FUNCTION_BLOCK CM_DoorLock EXTENDS CM_Base //--IMPLEMENTS I_Door
VAR_INPUT
	i_stSettings : ST_SettingsDoorLock;
END_VAR
VAR
	// Inputs
	I_bStaDoorIsClosed AT %I* : BOOL; // Door is closed
	I_bStaLockIsReleased AT %I* : BOOL; // Lock is released
	
	// Outputs
	Q_bCmdReleaseLock AT %Q* : BOOL; // FALSE = Apply, TRUE = Release
			
	// Requests
	s_bReqReleaseLock : BOOL;
	s_bReqApplyLock : BOOL;
	
	//----------------------Properties---------------------------//
	// States
	s_bStaDoorIsClosed : BOOL;
	s_bStaDoorIsOpened : BOOL;
	s_bStaLockIsApplied : BOOL;
	s_bStaLockIsReleased : BOOL;
	s_bCfgAutoLockAtClosing : BOOL;
	
	// Timers
	s_tonReleasingLockTimeout : TON;
	s_tonApplyingLockTimeout : TON;
	
	// Alarms
	s_fbAlarmHandlerReleasingLockTimeout : FB_AlarmHandler;
	s_fbAlarmHandlerApplyingLockTimeout : FB_AlarmHandler;
	s_fbAlarmHandlerDoorIsNotClosed : FB_AlarmHandler;
	
	s_errLockReleasingTimeout : BOOL;
	s_errLockApplyingTimeout : BOOL;
	s_wrnDoorIsNotClosed : BOOL;
		
	s_bStaDoorIsClosedOsr : R_TRIG; 
END_VAR


SUPER^();

METHOD PROTECTED _m_Alarms : BOOL

IF NOT SUPER^._m_Alarms() THEN
	RETURN;
END_IF

// Timeout (timers)
s_tonReleasingLockTimeout(
	IN := i_bReqEnable AND s_bReqReleaseLock AND NOT(s_bStaLockIsReleased),
	PT := i_stSettings.tReleasingLockTimeout);
	
s_tonApplyingLockTimeout(
	IN := i_bReqEnable AND s_bReqApplyLock AND NOT(s_bStaLockIsApplied),
	PT := i_stSettings.tApplyingLockTimeout);

// Set error bits
s_errLockReleasingTimeout := (s_tonReleasingLockTimeout.Q OR s_errLockReleasingTimeout) AND NOT(i_bCmdReset);
s_errLockApplyingTimeout := (s_tonApplyingLockTimeout.Q OR s_errLockApplyingTimeout) AND NOT(i_bCmdReset);

// Alarm Handlers
s_fbAlarmHandlerReleasingLockTimeout(
	i_bStaActive := s_errLockReleasingTimeout,
	i_eAlarmLevel := E_AlarmLevel.Alarm,
	i_sAlarmText := CONCAT(i_sCmName , ': Lock - releasing timeout.') );
	
s_fbAlarmHandlerApplyingLockTimeout(
	i_bStaActive := s_errLockApplyingTimeout,
	i_eAlarmLevel := E_AlarmLevel.Alarm,
	i_sAlarmText := CONCAT(i_sCmName , ': Lock - applying timeout.') );
	
s_fbAlarmHandlerDoorIsNotClosed(
	i_bStaActive := s_wrnDoorIsNotClosed,
	i_eAlarmLevel := E_AlarmLevel.Warning,
	i_sAlarmText := CONCAT(i_sCmName , ': Door - not closed (close door before lock can be applied).') );	
	
// Alarm collector	
s_bStaError := 
	s_fbAlarmHandlerReleasingLockTimeout.q_bStaActive
	OR s_fbAlarmHandlerApplyingLockTimeout.q_bStaActive;

_m_Alarms := TRUE;
END_METHOD

METHOD PROTECTED _m_Devices : BOOL

IF NOT SUPER^._m_Devices() THEN
	RETURN;
END_IF

IF s_bStaError THEN
	s_bReqReleaseLock := FALSE;
	s_bReqApplyLock := FALSE;
END_IF
	
IF s_bCfgAutoLockAtClosing AND s_bStaDoorIsClosedOsr.Q THEN
	s_bReqReleaseLock := FALSE;
	s_bReqApplyLock := TRUE;
END_IF

IF s_bStaDoorIsClosed THEN
	s_wrnDoorIsNotClosed := FALSE;	
END_IF

_m_Devices := TRUE;
END_METHOD

METHOD PROTECTED _m_Hmi : BOOL

IF NOT SUPER^._m_Hmi() THEN
	RETURN;
END_IF

_m_Hmi := TRUE;
END_METHOD

METHOD PROTECTED _m_Init : BOOL

IF NOT SUPER^._m_Init() THEN
	RETURN;
END_IF

_m_Init := TRUE;
END_METHOD

METHOD PROTECTED _m_Inputs : BOOL

IF NOT SUPER^._m_Inputs() THEN
	RETURN;
END_IF

s_bStaLockIsReleased := I_bStaLockIsReleased;
s_bStaLockIsApplied := NOT(I_bStaLockIsReleased);
s_bStaDoorIsClosed := I_bStaDoorIsClosed;
s_bStaDoorIsOpened := NOT(I_bStaDoorIsClosed);

s_bStaDoorIsClosedOsr(CLK := s_bStaDoorIsClosed);

_m_Inputs := TRUE;
END_METHOD

METHOD PROTECTED _m_Outputs : BOOL

IF NOT SUPER^._m_Outputs() THEN
	RETURN;
END_IF

Q_bCmdReleaseLock := s_bReqReleaseLock;

_m_Outputs := TRUE;
END_METHOD

/// Request to apply door-lock (only if door is closed)
METHOD PUBLIC m_Apply : BOOL

IF NOT i_bReqEnable THEN 
	RETURN;
END_IF

IF s_bStaDoorIsClosed THEN
	s_bReqReleaseLock := FALSE;
	s_bReqApplyLock := TRUE;
ELSE
	s_wrnDoorIsNotClosed := TRUE;	
END_IF
	
m_Apply := TRUE;
END_METHOD

/// Request to release door-lock
METHOD PUBLIC m_Release : BOOL

IF NOT i_bReqEnable THEN 
	RETURN;
END_IF

s_bReqReleaseLock := TRUE;
s_bReqApplyLock := FALSE;
s_wrnDoorIsNotClosed := FALSE;

m_Release := TRUE;
END_METHOD

{attribute 'monitoring':='call'}
PROPERTY PUBLIC p_bCfgAutoLockAtClosing : BOOL
GET

p_bCfgAutoLockAtClosing := s_bCfgAutoLockAtClosing;
END_GET
SET

s_bCfgAutoLockAtClosing := p_bCfgAutoLockAtClosing;
END_SET
END_PROPERTY

{attribute 'monitoring':='call'}
PROPERTY PUBLIC p_bStaDoorIsClosed : BOOL
GET

p_bStaDoorIsClosed := s_bStaDoorIsClosed;
END_GET
END_PROPERTY

{attribute 'monitoring':='call'}
PROPERTY PUBLIC p_bStaLockIsApplied : BOOL
GET

p_bStaLockIsApplied := s_bStaLockIsApplied;
END_GET
END_PROPERTY

{attribute 'monitoring':='call'}
PROPERTY PUBLIC p_bStaLockIsReleased : BOOL
GET

p_bStaLockIsReleased := s_bStaLockIsReleased;
END_GET
END_PROPERTY

END_FUNCTION_BLOCK

(* stored: Version 1.1.0.1, ProductVersion 3.1.4024.12
   POU CM_DoorLock: Id {ea68c333-cb10-44e9-998f-ee97a6acb23c}, SpecialFunc None
   Folder Methods: Id {f1e13262-5093-4e19-b253-1c3417c042de}
   Folder Properties: Id {1cd224f2-8e0f-4515-bca2-e2383476522d}
   Method _m_Alarms: Id {9c548875-33a6-42e4-a316-602892fa3d9c}
   Method _m_Devices: Id {610e92a2-55de-4c20-9dc9-5d6693ddaa6b}
   Method _m_Hmi: Id {099a1203-e422-4fa7-896f-2cb9acc72e21}
   Method _m_Init: Id {7e974ef6-a453-4752-8fef-bd0c78d3fc41}
   Method _m_Inputs: Id {0f80ea41-d213-4e61-bf55-0e2eaf7e039c}
   Method _m_Outputs: Id {505e11af-7bdd-44b3-8506-0a1a26a8e0b6}
   Method m_Apply: Id {1802c1c5-3d52-4491-b19a-2db94b292512}
   Method m_Release: Id {4b2987be-5b37-448a-ae60-0d85428f41cd}
   Property p_bCfgAutoLockAtClosing: Id {b297b3cd-a9e7-439b-828a-9dc922b1cecc}
   Get Get: Id {ebf2f841-0df8-4aa1-82c1-f182980d7fd3}
   Set Set: Id {d4466a48-d57f-43a1-b43f-4fc5b971cc4a}
   Property p_bStaDoorIsClosed: Id {6fc03739-dce9-4ee2-80bf-9e9172243c54}
   Get Get: Id {0a1b8b1e-e1eb-426d-a4e4-2cee32698ff0}
   Property p_bStaLockIsApplied: Id {30b69388-1c5c-4cc9-9c25-d58f841ab12c}
   Get Get: Id {2cd3b54e-5a1b-4a83-a32c-e86b48816fb2}
   Property p_bStaLockIsReleased: Id {ace57d84-4ff8-4d03-a4df-c730a29a90b7}
   Get Get: Id {25e3e480-7e08-4443-a7b7-3684820a84de} *)
